FUNCTION F_NormVec3 : LREAL
VAR_INPUT
    iVec3 : I_Vec3;
END_VAR


F_NormVec3 := SQRT(F_NormSqVec3(iVec3));

END_FUNCTION

(* stored: Version 1.1.0.1
   POU F_NormVec3: Id {d4ef8095-c2f1-4b9c-a3ce-569f407d34e8}, SpecialFunc None *)
